FUNCTION_BLOCK Stage5 (* Template for a Basic Function Block Type *)
  (* Standard: 61499-2 *)
  (* Version 1.0, 2021-06-20, HP *)
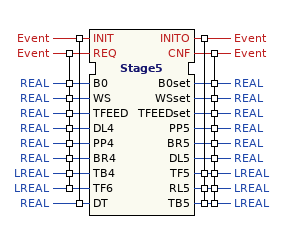
  EVENT_INPUT
    INIT WITH DT; (* Initialization Request *)
    REQ WITH B0, WS, TFEED, DL4, PP4, BR4, TB4, TF6; (* Normal Execution Request *)
  END_EVENT
  EVENT_OUTPUT
    INITO WITH TB5, RL5, TF5; (* Initialization Confirm *)
    CNF WITH TB5, DL5, TF5, BR5, PP5, RL5, B0set, WSset, TFEEDset; (* Execution Confirmation *)
  END_EVENT
  VAR_INPUT
    B0 : REAL;
    WS : REAL;
    TFEED : REAL;
    DL4 : REAL;
    PP4 : REAL;
    BR4 : REAL;
    TB4 : LREAL;
    TF6 : LREAL;
    DT : REAL;
  END_VAR
  VAR_OUTPUT
    B0set : REAL;
    WSset : REAL;
    TFEEDset : REAL;
    PP5 : REAL;
    BR5 : REAL;
    DL5 : REAL;
    TF5 : LREAL;
    RL5 : LREAL;
    TB5 : LREAL;
  END_VAR
  VAR
    AB : REAL; (* internal variabel *)
    UU : REAL;
    TREF : REAL;
    AD : REAL;
    AHC : REAL;
    AHR : REAL;
    AS : REAL;
    REC : REAL;
    WN : REAL;
    WN_1 : REAL;
    XKN : REAL;
    C1 : REAL;
    HS : REAL;
    G : REAL;
    W1 : REAL;
    TFREC : REAL;
    TS : REAL;
    DTS : REAL;
    TF5_last : REAL;
    RL5_last : REAL;
    TB5_last : REAL;
    USS : REAL;
    RHOB : REAL;
    CPB : REAL;
    CPF : REAL;
    FMW : REAL;
    HLV : REAL;
    HV : REAL;
    BPR : REAL;
    FMC : REAL;
    U : REAL;
    A : REAL;
    B : REAL;
    C : REAL;
    D1 : REAL;
    d : REAL;
    a : REAL;
    A1 : REAL;
    A2 : REAL;
    A3 : REAL;
    A4 : REAL;
    A5 : REAL;
    A6 : REAL;
    p : REAL;
    q : REAL;
    TC : REAL;
    PC : REAL;
    DTB5 : REAL;
    DEN5 : REAL;
    DH5 : REAL;
    DP5 : REAL;
    DPDH5 : REAL;
    DT5 : REAL;
    m : REAL;
    n : REAL;
    VR5 : REAL;
    DELTA5 : REAL;
    DELTA27 : REAL;
    DELTA49 : REAL;
    DELTA5_last : REAL;
    DELTA27_last : REAL;
    DELTA49_last : REAL;
  END_VAR
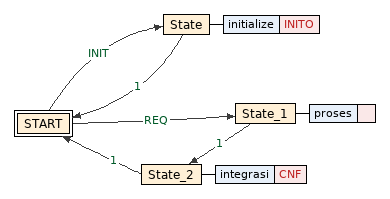
  EC_STATES
    START; (* Initial State *)
    State : initialize -> INITO;
    State_1 : proses;
    State_2 : integrasi -> CNF;
  END_STATES
  EC_TRANSITIONS
    START TO State := INIT;
    State TO START := 1;
    START TO State_1 := REQ;
    State_1 TO State_2 := 1;
    State_2 TO START := 1;
  END_TRANSITIONS
  ALGORITHM initialize IN ST: (* Initialization algorithm *)
TREF :=273.15;
AB :=57.2727;
AHC :=4069.2;
AHR :=2639.7;
AS :=3225.7;
REC :=0.0;
//TF2:=TF2;

//TFEED :=TFEED1+TREF;
 //TS:=TS1+TREF;
WN :=3.0;
XKN :=0.68;
HS:=0.11;
G :=9.81;
W1 :=0.50;

RL5 := 0.539427232788953;
TB5 := 353.681541592948;
TF5 := 349.772691418052;
TF6 := 347.148389575489;



RL5_last :=RL5;
TB5_last :=TB5;
TF5_last :=TF5;
  END_ALGORITHM
  ALGORITHM proses IN ST: (* kalkulasi *)
UU := TFEED;
U :=UU;

USS :=49.767;
C1 :=0.625;
RHOB :=1032.4; //maassa jenis brine
CPB :=1.00; //heatcapacity Brine
CPF :=1.00; //heat capacity feed
FMW :=23654.0;
HLV :=563.7959;
HV :=625.1971;
BPR :=2.192;
FMC :=34736.09;
//U :=UU; //feed temp



///  Calculate the physical properties

//A :=3.2437814;
//B :=5.86826*0.001;
//C :=1.1702379*0.00000001;
//D1 :=2.1878462*0.001;
//TC :=647.27;
//PC :=218.167;


A1 :=3.2437814;
A2:=5.86826*0.001;
A3:=1.1702379*0.00000001;
A4 :=2.1878462*0.001;
A5 :=647.27;
A6 :=218.167;

DTB5 :=A5-TB5;
DEN5 :=(A1+A2*DTB5+A3*DTB5*DTB5*DTB5)/(1+A4*DTB5)*DTB5/TB5;
p:=DEN5;
q:=10.0;
PP5 :=A6/(EXPT(q, p));

// calculate the brine flow rates
DP5:=PP4-PP5;
DH5:=RL5-C1*HS;
DPDH5 :=DP5*101000+G*RHOB*DH5;
m:=DPDH5*RHOB;
n:=0.5;
BR5 :=WN*XKN*RL5*(EXPT(m, n));
BR5 :=BR5*60.0/1000.0;

// calculate the vapor flow rates

DT5 :=TB5-BPR/1.8-(TF6+TF5)*0.5;
VR5 :=U*AHC*DT5/HLV/1000.0;
DL5 :=DL4+VR5;


//// state equation
DELTA5 :=(BR4-BR5-VR5)*1000.0/RHOB/AB;
DELTA27 :=((BR4*CPB*(TB4-TB5))-VR5*(HV-CPB*(TB5-TREF)))*1000.0/AB/RHOB/CPB/RL5;
DELTA49 :=((B0*CPF*(TF6-TF5)*1000+(U*AHC*DT5)))/FMW/CPF;
  END_ALGORITHM
  ALGORITHM integrasi IN ST: (* new algorithm *)
B0set:=B0;
WSset:=WS ;
TFEEDset:=TFEED;
//integrasi
RL5 := (DELTA5 + DELTA5_last)*0.5*DT + RL5_last;
DELTA5_last :=DELTA5 ;
RL5_last :=RL5;

TB5 := (DELTA27 + DELTA27_last)*0.5*DT + TB5_last;
DELTA27_last :=DELTA27 ;
TB5_last:=TB5;

TF5 := (DELTA49 + DELTA49_last)*0.5*DT + TF5_last;
DELTA49_last :=DELTA49 ;
TF5_last :=TF5;
  END_ALGORITHM
END_FUNCTION_BLOCK
